{attribute 'qualified_only'}
VAR_GLOBAL
END_VAR

(* stored: Version 1.1.0.1, ProductVersion 3.1.4022.7
   GVL GVL_02_Parameter_Servo_Motor_Robot: Id {a0bb10da-edf9-4d69-9305-2e33817f70dd} *)
